// TIA Portal V17 export
// export: Created 2026-04-13T11:12:44.3830945Z, ExportSetting WithDefaults, DisplayName Totally Integrated Automation Portal, DisplayVersion V17 Update 4, DisplayName TIA Portal Openness, DisplayVersion V17 Update 4, DisplayName TIA Portal Version Control Interface, DisplayVersion V17, DisplayName SINAMICS Startdrive Advanced, DisplayVersion V17, DisplayName SINAMICS Startdrive G130, G150, S120, S150, SINAMICS MV, S210, DisplayVersion V17, DisplayName SINAMICS Startdrive G110M, G120, G120C, G120D, G120P, G115D, DisplayVersion V17, DisplayName STEP 7 Professional, DisplayVersion V17 Update 4, DisplayName STEP 7 Safety, DisplayVersion V17, DisplayName WinCC Professional, DisplayVersion V17 Update 4
DATA_BLOCK "A5-模拟量输出_DB"   // DB11
VERSION : 0.1
// stored: AutoNumber true, DBAccessibleFromOPCUA true, DBAccessibleFromWebserver true, InstanceOfName A5-模拟量输出, InstanceOfType FB
"A5-模拟量输出"
   // VAR
   //    进风加热比例调节阀 { S7_SetPoint := 'True'} : "A2-数据转换RTI";
   //    回风加热比例调节阀 { S7_SetPoint := 'True'} : "A2-数据转换RTI";
   //    放空比例调节阀 { S7_SetPoint := 'True'} : "A2-数据转换RTI";
   // END_VAR
BEGIN
END_DATA_BLOCK
